TYPE ST_ServerResponse :
STRUCT
	nStatus     : INT;
    fValue      : REAL;
    nErrorCode  : INT;
END_STRUCT
END_TYPE

(* stored: Version 1.1.0.1, ProductVersion 3.1.4024.16
   DUT ST_ServerResponse: Id {16ea6d8f-8598-442a-a821-d21170d4a9b4} *)
